Staubli VAL3: pp_bs_f1f2f3.pgx

program pp_bs_f1f2f3()
begin
  //given f1,f2,f3 are in hand
  //exit state : f1,f2,f3 secured in bs

  //place f2 in origin of bk (//open bk vacuum
  call regular_place(t1,mNomSpeed,mSlowSpeed,pPointRx_f1_bk,false,dDio_t1_cy,true)

  //place f2 in origin of bk (//open bk vacuum
  call regular_place(t2,mNomSpeed,mSlowSpeed,pPointRx_f2_bk,false,dDio_t2_cy,true)

  //drop f3 offset from f2 origin
  call regular_place(t3,mNomSpeed,mSlowSpeed,pPointRx_f3_bk,false,dDio_t3_cy,true)

end
